FUNCTION_BLOCK FB_Metalization
VAR_INPUT
	ins_CommIn		: Type_CommIn_Metalization;
END_VAR
VAR_OUTPUT
	outs_CommOut	: Type_CommOut_Metalization;
	o_Read			:BOOL;
END_VAR
VAR
	o_TotalCycleTime	:BYTE;
	o_PartExists AT %Q*	:BOOL;
	o_ProcessCycleTime	AT %Q*		:BYTE;
	
	RetVal : enum_RetVal;
	
	(* Timers *)
	
	T01_Init_Metalization		:TON;
	T02_Check_Part_Here			:TON;
	T03_Check_Chemical			:TON;
	T04_Add_To_Bath				:TON;
	T05_Remove_From_Bath		:TON;
	T06_Check_Robot_Here		:TON;
	T07_Return_Part				:TON;
	
	Instance_CountTotalCycleTime		:FB_CountCycleTime();
	Instance_CountProcessCycleTime		:FB_CountCycleTime();
	
END_VAR

A01_AutomaticMode();

ACTION A01_AutomaticMode:
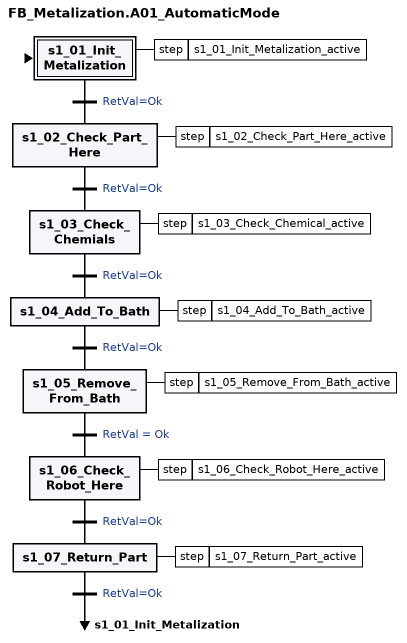
INITIAL_STEP s1_01_Init_Metalization:
    s1_01_Init_Metalization_active(N);  // step action
END_STEP
TRANSITION FROM s1_01_Init_Metalization TO s1_02_Check_Part_Here
    := RetVal=Ok;
END_TRANSITION
STEP s1_02_Check_Part_Here:
    s1_02_Check_Part_Here_active(N);  // step action
END_STEP
TRANSITION FROM s1_02_Check_Part_Here TO s1_03_Check_Chemials
    := RetVal=Ok;
END_TRANSITION
STEP s1_03_Check_Chemials:
    s1_03_Check_Chemical_active(N);  // step action
END_STEP
TRANSITION FROM s1_03_Check_Chemials TO s1_04_Add_To_Bath
    := RetVal=Ok;
END_TRANSITION
STEP s1_04_Add_To_Bath:
    s1_04_Add_To_Bath_active(N);  // step action
END_STEP
TRANSITION FROM s1_04_Add_To_Bath TO s1_05_Remove_From_Bath
    := RetVal=Ok;
END_TRANSITION
STEP s1_05_Remove_From_Bath:
    s1_05_Remove_From_Bath_active(N);  // step action
END_STEP
TRANSITION FROM s1_05_Remove_From_Bath TO s1_06_Check_Robot_Here
    := RetVal = Ok;
END_TRANSITION
STEP s1_06_Check_Robot_Here:
    s1_06_Check_Robot_Here_active(N);  // step action
END_STEP
TRANSITION FROM s1_06_Check_Robot_Here TO s1_07_Return_Part
    := RetVal=Ok;
END_TRANSITION
STEP s1_07_Return_Part:
    s1_07_Return_Part_active(N);  // step action
END_STEP
TRANSITION FROM s1_07_Return_Part TO s1_01_Init_Metalization
    := RetVal=Ok;
END_TRANSITION
END_ACTION

ACTION s1_01_Init_Metalization_active:
RetVal:=Running;

Instance_CountTotalCycleTime(inm_TimeActive:=FALSE);
o_TotalCycleTime:=REAL_TO_BYTE(Instance_CountTotalCycleTime.outr_CycleTime);

outs_CommOut.s_Robot.m_Empty:=TRUE;
outs_CommOut.s_Robot.m_Ready:=FALSE;

IF ins_CommIn.s_Robot.m_OutOfArea
	THEN
	Instance_CountTotalCycleTime(inm_TimeActive:=TRUE);
	RetVal:=Ok;
END_IF
END_ACTION

ACTION s1_02_Check_Part_Here_active:
RetVal:=Running;

IF ins_CommIn.s_Robot.m_OutOfArea = FALSE(*Daca position[2] e true inseamna ca robotul e in pozitie, dar nu s-a facut place!!	*)
	AND ins_CommIn.s_Robot.m_Work = FALSE	
	THEN
	outs_CommOut.s_Robot.m_Empty:=FALSE;	
END_IF

IF ins_CommIn.s_Robot.m_PartDropped
	THEN
	RetVal:=Ok;
END_IF
END_ACTION

ACTION s1_03_Check_Chemical_active:
RetVal:=Running;

T03_Check_Chemical(IN:=TRUE,PT:=T#15S,Q=>,ET=>);

IF T03_Check_Chemical.Q
	THEN
	T03_Check_Chemical(IN:=FALSE);
	RetVal:=Ok;
END_IF
END_ACTION

ACTION s1_04_Add_To_Bath_active:
RetVal:=Running;

T04_Add_To_Bath(IN:=TRUE,PT:=T#5S,Q=>,ET=>);

IF T04_Add_To_Bath.Q
	THEN
	T04_Add_To_Bath(IN:=FALSE);
	RetVal:=Ok;
END_IF
END_ACTION

ACTION s1_05_Remove_From_Bath_active:
RetVal:=Running;

T05_Remove_From_Bath(IN:=TRUE,PT:=T#5S,Q=>,ET=>);

IF T05_Remove_From_Bath.Q
	THEN
	Instance_CountProcessCycleTime(inm_TimeActive:=FALSE);
	o_ProcessCycleTime:=REAL_TO_BYTE(Instance_CountProcessCycleTime.outr_CycleTime);
	
	outs_CommOut.s_Robot.m_Ready:=TRUE;
	T05_Remove_From_Bath(IN:=FALSE);
	RetVal:=Ok;
END_IF
END_ACTION

ACTION s1_06_Check_Robot_Here_active:
RetVal:=Ok;
END_ACTION

ACTION s1_07_Return_Part_active:
RetVal:=Running;

T07_Return_Part(IN:=TRUE,PT:=T#5S,Q=>,ET=>);

o_PartExists:=FALSE;

IF T07_Return_Part.Q
	THEN
	Global_Vars.NoOfPartsDone:=Global_Vars.NoOfPartsDone + 1;
	T07_Return_Part(IN:=FALSE);
	RetVal:=Ok;
END_IF
END_ACTION

END_FUNCTION_BLOCK

(* stored: Version 1.1.0.1, ProductVersion 3.1.4024.3
   POU FB_Metalization: Id {77e26e9f-bbfe-4123-9612-62be36e9d3cc}, SpecialFunc None
   Folder S1: Id {20a24cce-96cb-4d03-9c8d-082b466a3a6f}
   Folder S2: Id {02341d1f-6004-49ef-8323-6f454676d28c}
   Action A01_AutomaticMode: Id {7e6a3ab1-335e-46d9-9aeb-ca273d9e7969}
   Action s1_01_Init_Metalization_active: Id {0e021d88-cb6c-4535-865b-de563f6341a8}
   Action s1_02_Check_Part_Here_active: Id {505fade0-2e4f-4cdf-8d87-4d03796192ef}
   Action s1_03_Check_Chemical_active: Id {d6ecaa08-0cc1-485a-b2d6-93de4a2b5545}
   Action s1_04_Add_To_Bath_active: Id {860a52c7-18a3-4fb3-8fee-e0ad34d8284b}
   Action s1_05_Remove_From_Bath_active: Id {a8a0f80b-b830-41ad-8f00-c1731c68d14e}
   Action s1_06_Check_Robot_Here_active: Id {fd3528bd-9b06-4f44-9ee7-ba20c2a79fb3}
   Action s1_07_Return_Part_active: Id {690759b8-777d-4829-b5c6-daeefa349d89} *)
